TYPE ref_ele_output :
STRUCT
	out_flg_eleA : BOOL;
	out_flg_eleB : BOOL;
	out_flg_reset : BOOL;
END_STRUCT
END_TYPE

(* stored: Version 1.1.0.1, ProductVersion 3.1.4024.11
   DUT ref_ele_output: Id {0eed964e-56f8-49c5-b6fd-f46d15160d32} *)
